PROGRAM VltSplit
VAR
	t1 : TON;
	a : BOOL;
	pt : TIME;
	done : BOOL;
END_VAR

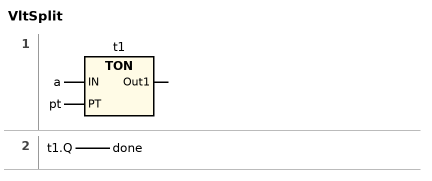
// NETWORK 1
t1(IN := a, PT := pt); // TON

// NETWORK 2
done := t1.Q;

END_PROGRAM

(* stored: Version 1.1.0.1, ProductVersion 3.1.4024.16
   POU VltSplit: Id {7dee3d69-3dfc-4528-a928-b54459e36e5b}, SpecialFunc None *)
